(* IEC 61131-3 sources: Study-OpenPLC/prog_Counter/build, 2 files *)

(* ---- plc.st ---- *)
TYPE
  LOGLEVEL : (CRITICAL, WARNING, INFO, DEBUG) := INFO;
END_TYPE

FUNCTION_BLOCK LOGGER
  VAR_INPUT
    TRIG : BOOL;
    MSG : STRING;
    LEVEL : LOGLEVEL := INFO;
  END_VAR
  VAR
    TRIG0 : BOOL;
  END_VAR

  IF TRIG AND NOT TRIG0 THEN
  {{
   LogMessage(GetFbVar(LEVEL),(char*)GetFbVar(MSG, .body),GetFbVar(MSG, .len));
  }}
  END_IF;
  TRIG0:=TRIG;
END_FUNCTION_BLOCK

FUNCTION_BLOCK python_eval
  VAR_INPUT
    TRIG : BOOL;
    CODE : STRING;
  END_VAR
  VAR_OUTPUT
    ACK : BOOL;
    RESULT : STRING;
  END_VAR
  VAR
    STATE : DWORD;
    BUFFER : STRING;
    PREBUFFER : STRING;
    TRIGM1 : BOOL;
    TRIGGED : BOOL;
  END_VAR

  {extern void __PythonEvalFB(int, PYTHON_EVAL*);__PythonEvalFB(0, data__);}
END_FUNCTION_BLOCK

FUNCTION_BLOCK python_poll
  VAR_INPUT
    TRIG : BOOL;
    CODE : STRING;
  END_VAR
  VAR_OUTPUT
    ACK : BOOL;
    RESULT : STRING;
  END_VAR
  VAR
    STATE : DWORD;
    BUFFER : STRING;
    PREBUFFER : STRING;
    TRIGM1 : BOOL;
    TRIGGED : BOOL;
  END_VAR

  {extern void __PythonEvalFB(int, PYTHON_EVAL*);__PythonEvalFB(1,(PYTHON_EVAL*)(void*)data__);}
END_FUNCTION_BLOCK

FUNCTION_BLOCK python_gear
  VAR_INPUT
    N : UINT;
    TRIG : BOOL;
    CODE : STRING;
  END_VAR
  VAR_OUTPUT
    ACK : BOOL;
    RESULT : STRING;
  END_VAR
  VAR
    py_eval : python_eval;
    COUNTER : UINT;
    _TMP_ADD10_OUT : UINT;
    _TMP_EQ13_OUT : BOOL;
    _TMP_SEL15_OUT : UINT;
    _TMP_AND7_OUT : BOOL;
  END_VAR

  _TMP_ADD10_OUT := ADD(COUNTER, 1);
  _TMP_EQ13_OUT := EQ(N, _TMP_ADD10_OUT);
  _TMP_SEL15_OUT := SEL(_TMP_EQ13_OUT, _TMP_ADD10_OUT, 0);
  COUNTER := _TMP_SEL15_OUT;
  _TMP_AND7_OUT := AND(_TMP_EQ13_OUT, TRIG);
  py_eval(TRIG := _TMP_AND7_OUT, CODE := CODE);
  ACK := py_eval.ACK;
  RESULT := py_eval.RESULT;
END_FUNCTION_BLOCK

PROGRAM prog
  VAR
    Plus : BOOL;
  END_VAR
  VAR
    LED : INT;
  END_VAR
  VAR
    Reset : BOOL;
    SetTime : TIME := T#100ms;
    Counter : INT;
    MaxValue : INT := 255;
    CTU0 : CTU;
    TON0 : TON;
    TOF0 : TOF;
    R_TRIG1 : R_TRIG;
  END_VAR

  TON0(IN := NOT(Plus), PT := SetTime);
  TOF0(EN := TON0.ENO, IN := TON0.Q, PT := SetTime);
  Plus := TOF0.Q;
  LED := Counter;
  R_TRIG1(CLK := Plus);
  CTU0(CU := R_TRIG1.Q, R := Reset, PV := MaxValue);
  Counter := CTU0.CV;
END_PROGRAM

CONFIGURATION Config0

  RESOURCE Res0 ON PLC
    TASK task0(INTERVAL := T#20ms,PRIORITY := 0);
    PROGRAM instance0 WITH task0 : prog;
  END_RESOURCE
END_CONFIGURATION

(* ---- generated_plc.st ---- *)
PROGRAM prog
  VAR
    Plus : BOOL;
  END_VAR
  VAR
    LED AT %QX0.0 : INT;
  END_VAR
  VAR
    Reset : BOOL;
    SetTime : TIME := T#100ms;
    Counter : INT;
    MaxValue : INT := 255;
    CTU0 : CTU;
    TON0 : TON;
    TOF0 : TOF;
    R_TRIG1 : R_TRIG;
  END_VAR

  TON0(IN := NOT(Plus), PT := SetTime);
  TOF0(EN := TON0.ENO, IN := TON0.Q, PT := SetTime);
  Plus := TOF0.Q;
  LED := Counter;
  R_TRIG1(CLK := Plus);
  CTU0(CU := R_TRIG1.Q, R := Reset, PV := MaxValue);
  Counter := CTU0.CV;
END_PROGRAM

CONFIGURATION Config0

  RESOURCE Res0 ON PLC
    TASK task0(INTERVAL := T#20ms,PRIORITY := 0);
    PROGRAM instance0 WITH task0 : prog;
  END_RESOURCE
END_CONFIGURATION
